PROGRAM DoSomeMath
VAR_INPUT
	i_rInputA: REAL;
	i_rInputB: REAL;
END_VAR
VAR
END_VAR

END_PROGRAM

(* stored: Version 1.1.0.1, ProductVersion 3.1.4022.12
   POU DoSomeMath: Id {09824f07-72e5-4c56-b34e-7785a772a76b}, SpecialFunc None *)
